{attribute 'qualified_only'}
VAR_GLOBAL
	Axes		: ARRAY[0..4] OF FB_Axis;
	AxesFaults	: ARRAY[0..4] OF ST_AxisFault;
END_VAR

(* stored: Version 1.1.0.1, ProductVersion 3.1.4024.12
   GVL GVL: Id {712c2e96-15a0-4761-b30c-03108217af0d} *)
